INTERFACE I_RpcServer

METHOD PUBLIC GetConfiguredHeaderSize : UDINT
VAR_INPUT
END_VAR
END_METHOD

METHOD PUBLIC GetConfiguredPayloadSize : UDINT
VAR_INPUT
END_VAR
END_METHOD

{attribute 'TcRpcEnable'}
METHOD PUBLIC HandleRequest : ResponseData;
VAR_INPUT
	SerializedHeader : STRING(ServerConfiguration.HEADER_STRING_SIZE);
	SerializedPayload : STRING(ServerConfiguration.PAYLOAD_STRING_SIZE);
END_VAR
END_METHOD

METHOD PUBLIC RegisterApi
VAR_INPUT
	RpcApi : I_RpcApi;
END_VAR
END_METHOD

METHOD PUBLIC RegisterAsynchronousRpcHandler
VAR_INPUT
	MethodName : T_MAXSTRING;
	Handler : I_AsynchronousRpcHandler;
END_VAR
END_METHOD

METHOD PUBLIC RegisterSynchronousRpcHandler
VAR_INPUT
	MethodName : T_MAXSTRING;
	Handler : I_SynchronousRpcHandler;
END_VAR
END_METHOD

END_INTERFACE

(* stored: Version 1.1.0.1, ProductVersion 3.1.4024.13
   Itf I_RpcServer: Id {3249790d-2361-4909-9f7a-771c2ba70619}
   Method GetConfiguredHeaderSize: Id {52438743-34c7-4348-a43a-8f0da9e009a4}
   Method GetConfiguredPayloadSize: Id {9c82b554-227f-4316-99a8-63da45a2124e}
   Method HandleRequest: Id {030ecb1b-b923-49ad-bdf9-2ab33a6cffbf}
   Method RegisterApi: Id {1683fa06-5bc8-42bf-97be-84865033b985}
   Method RegisterAsynchronousRpcHandler: Id {c7ede9aa-6e51-466a-80ea-5a4569d1c9eb}
   Method RegisterSynchronousRpcHandler: Id {e9370da5-05df-4cae-8260-53b6cf2d257e} *)
